// SIMATIC S7-200 SMART project (STEP 7-Micro/WIN SMART), CPU SR40

SYMBOL_TABLE 用户定义1
字符2              'DCBA'
字符串1             "ABCDE"
END_SYMBOL_TABLE

ORGANIZATION_BLOCK 主程序:OB1
TITLE=程序注释
BEGIN
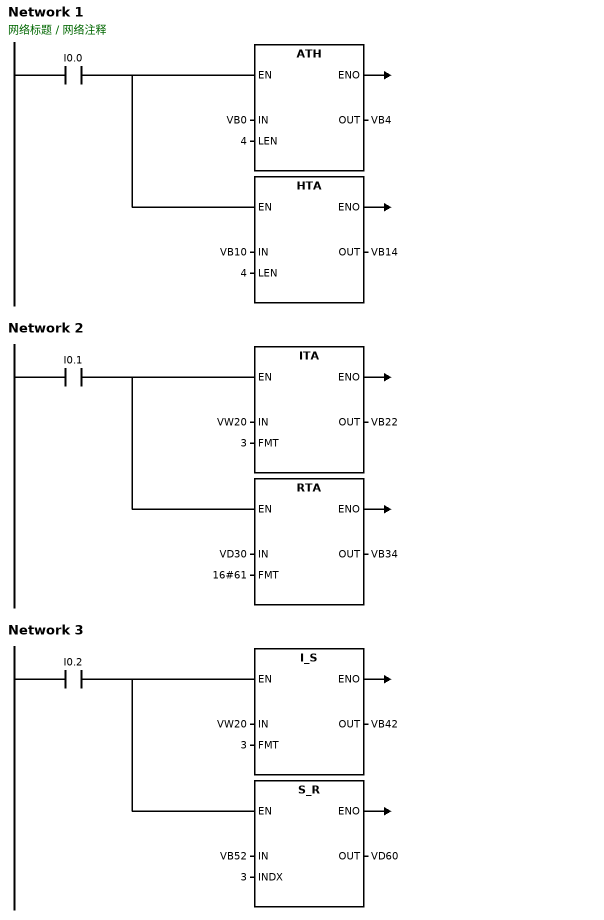
Network 1
// 网络标题
// 网络注释
LD     I0.0
ATH    VB0, VB4, 4
HTA    VB10, VB14, 4
Network 2
LD     I0.1
ITA    VW20, VB22, 3
RTA    VD30, VB34, 16#61
Network 3
LD     I0.2
ITS    VW20, VB42, 3
?2B2   VB52, 3, VD60
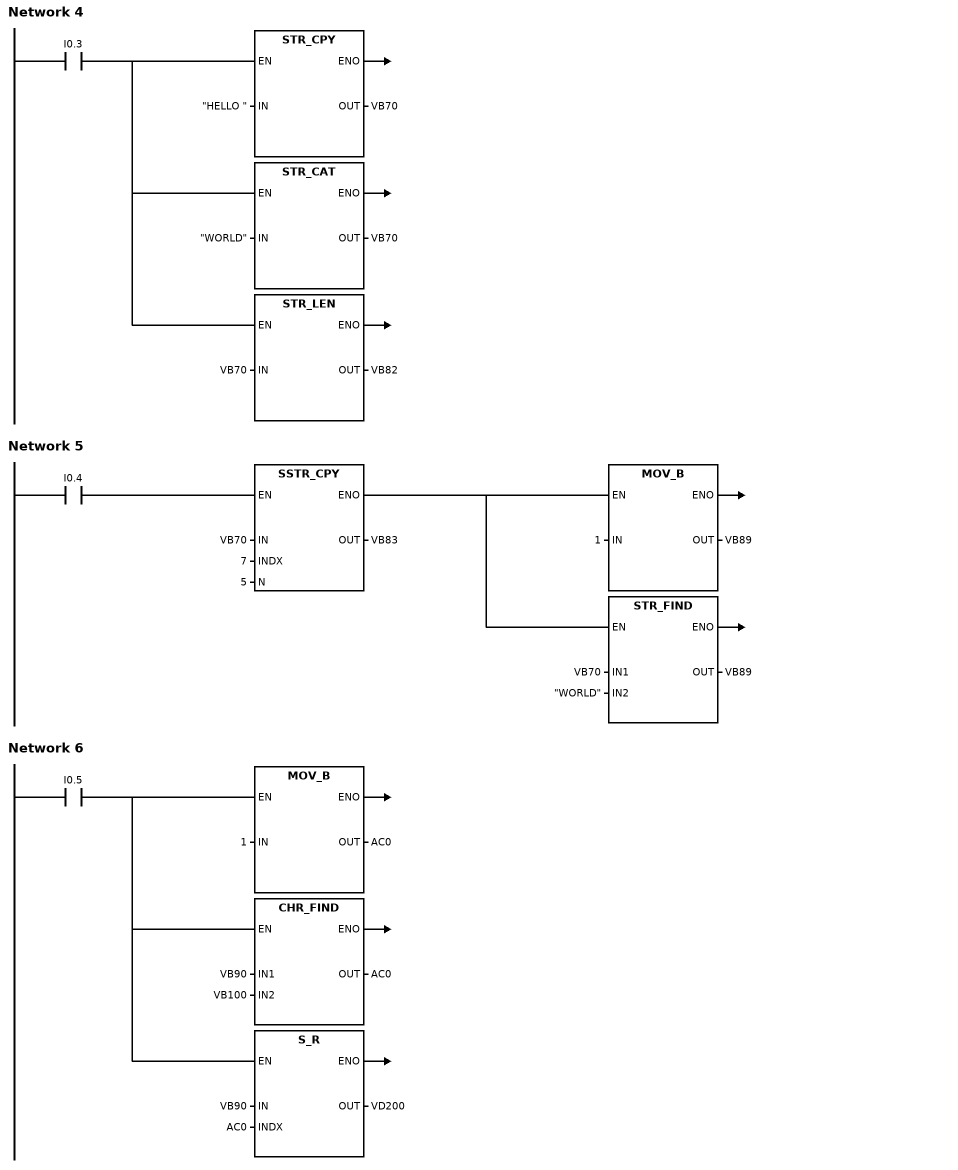
Network 4
//将字符串"HELLO "复制到VB70开始的存储区
//将字符串"WORLD"附到VB70开始的字符串的后面
//求VB70开始的字符串的长度
LD     I0.3
SCPY   "HELLO ", VB70
SCAT   "WORLD", VB70
SLEN   VB70, VB82
Network 5
LD     I0.4
SSCPY  VB70, 7, 5, VB83
AENO
MOVB   1, VB89
SFND   VB70, "WORLD", VB89
Network 6
//AC0用作OUT参数并指向字符串的首个字符。
//在VB90开始的字符串中寻找数字字符
//将字符串中的温度值转换为实数
LD     I0.5
MOVB   1, AC0
CFND   VB90, VB100, AC0
?2B2   VB90, AC0, VD200
END_ORGANIZATION_BLOCK

DATA_BLOCK_TAB 用户定义1
BEGIN
//数据页注释
//按 F1 键获取帮助和示范数据页
VB0      '3EA8'
VW10     16#2A38
VW20     -12345
VD30     -12.43
VB52     "V=123.4"
VB90     "T=239.8"
VB100    "1234567890+-"
END_DATA_BLOCK_TAB
